Staubli VAL3: HOME.pjx

--- HOME.pjx ---
Parameters version=s7.5.3 stackSize=5000 millimeterUnit=true
Program file=copy_it.pgx
Program file=link_it.pgx
Data file=HOME.dtx
Type name=TrajHome path=Disk://kernel/template/TrajHome/TrajHome.pjx

--- HOME.dtx ---
public TrajHome tTraj{}
  [home]
    num nIndexTool
    TrajJointItem tData
      [0]
        jointRx jJoint
        TrajectoryItem tSuper
          [0]
            num distance
            num moveType
            num nTime
            num nStop
            num nTcpAction
            string comment
            bool toStop
            mdesc nom_speed = {vel=50, tmax=500}
            InstrItem iInstr[3]
              [0]
                string sType
                string sData
              [1]
                string sType
                string sData
              [2]
                string sType
                string sData
            num nMoveId
    string sID = "home"
    num nZoneType
    num nZoneMove
    pointRx pO = {fatherId=world[0]}
    pointRx pX = {fatherId=world[0]}
    pointRx pY = {fatherId=world[0]}
    num nDimension
    pointRx pPointMove = {fatherId=tTraj["home"].fFrame[0]}
    frame fFrame = {fatherId=world[0]}
    string sProgram
    num nIndexFrame

--- copy_it.pgx ---
public program copy_it(string x_sCopy, string x_sPaste)
begin
  // try to copy it
  if isDefined(tTraj[x_sCopy])
    // copy it
    tTraj[x_sPaste]=tTraj[x_sCopy]
    //
  endIf
end
